(* CoDeSys 2.3 export: CLIENT_ACCEPT.EXP *)

(* Data type *)
TYPE CLIENT_ACCEPT :
STRUCT
	diSocket:DINT;
	stIPAddress:STRING(20);
END_STRUCT
END_TYPE
